# EPICS substitutions: ek9000App/Db/EL1124_mbbiDirect.substitutions
file EL1124.template
{       pattern
        {
                TERMINAL,

        }
        {
        }
}
